Yaskawa INFORM job: OK_R2_O26(120,90)POSPAWANE.JBI

/JOB
//NAME OK_R2_O26(120,90)POSPAWANE
///FOLDERNAME X4
//POS
///NPOS 76,76,76,3,0,0
///TOOL 0
///POSTYPE PULSE
///PULSE
C00000=-124687,-83177,-100814,4913,99770,76656
C00001=-124710,-87372,-98535,4861,96226,76509
C00002=-124720,-88823,-97522,4846,94862,76452
C00003=-124678,-87356,-95828,4839,94572,76455
C00004=-124720,-88823,-97522,4846,94862,76452
C00005=-94650,-94699,-99032,-20051,93372,70764
C00006=-96283,-95826,-99477,-19873,92695,70300
C00007=-94650,-94699,-99032,-20051,93372,70764
C00008=-127024,-94781,-101034,6932,94604,73639
C00009=-125486,-94406,-100478,6779,94328,74137
C00010=-125580,-97568,-101093,6774,93098,74039
C00011=-125486,-94406,-100478,6779,94328,74137
C00012=-127024,-94781,-101034,6932,94604,73639
C00013=-126741,-87687,-96957,6922,95710,73795
C00014=-126718,-86230,-97962,6944,97065,73878
C00015=-126662,-82027,-100223,7023,100586,74095
C00016=-123675,-116589,-109803,7997,69973,-81393
C00017=-122744,-114748,-105092,7760,67947,-81192
C00018=-122375,-113926,-103174,7667,67160,-81109
C00019=-124288,-113805,-103134,8357,67388,-81794
C00020=-124245,-111702,-101340,8343,67360,-81780
C00021=-124288,-113805,-103134,8357,67388,-81794
C00022=-122375,-113926,-103174,7667,67160,-81109
C00023=-138630,-81193,-91554,22902,91021,-82706
C00024=-137093,-81891,-91862,22646,90453,-82269
C00025=-138630,-81193,-91554,22902,91021,-82706
C00026=-138527,-80465,-90405,22879,90685,-82733
C00027=-99714,-84314,-92829,-14326,90379,-83348
C00028=-99332,-87085,-93392,-14378,89399,-83105
C00029=-99714,-84314,-92829,-14326,90379,-83348
C00030=-100119,-76546,-91010,-14307,93097,-83800
C00031=-99872,-75926,-91520,-14362,93752,-83793
C00032=-120615,-96879,-94500,12422,61763,-56469
C00033=-120615,-96444,-91045,12645,59903,-56681
C00034=-120614,-96198,-89632,12739,59177,-56766
C00035=-120612,-97964,-91396,12715,59351,-56744
C00036=-122358,-96168,-89622,13602,59468,-57423
C00037=-120614,-96100,-89110,12773,58912,-56797
C00038=-120614,-95936,-88283,12829,58498,-56846
C00039=-120614,-95844,-87846,12859,58281,-56872
C00040=-120614,-95993,-88552,13310,59748,-59437
C00041=-120614,-96276,-90020,13213,60486,-59348
C00042=-120615,-96798,-93612,12981,62380,-59123
C00043=-120616,-96853,-99747,5843,73141,-72527
C00044=-120615,-96881,-95746,5920,70677,-72647
C00045=-120615,-96762,-94095,5954,69726,-72694
C00046=-120646,-98510,-95846,5959,69908,-72696
C00047=-120787,-94368,-93966,5976,70884,-72697
C00048=-120615,-96784,-94531,4240,70392,-75290
C00049=-120615,-96741,-94529,-89,69852,-81815
C00050=-120615,-96737,-94499,-2085,69975,-84977
C00051=-120615,-96736,-94490,-2287,69985,-85289
C00052=-120615,-96833,-96173,-2273,70970,-85308
C00053=-120616,-96725,-100243,-2243,73529,-85356
C00054=-120616,-95180,-99735,-2469,75570,69309
C00055=-120615,-95387,-95787,-2498,73036,69361
C00056=-120615,-95334,-94154,-2510,72060,69381
C00057=-120451,-92546,-93661,-2552,73193,69414
C00058=-120612,-97039,-95899,-2509,72258,69378
C00059=-120615,-95352,-94373,-2037,72369,71923
C00060=-120615,-95364,-94077,-88,70775,81896
C00061=-120615,-95363,-94184,611,71183,86811
C00062=-120615,-95363,-94196,663,71233,87105
C00063=-120615,-95421,-95866,660,72230,87111
C00064=-120616,-95208,-99899,652,74822,87124
C00065=-120615,-95299,-94637,-6871,62387,55584
C00066=-120614,-95009,-91097,-7001,60372,55709
C00067=-120614,-94810,-89647,-7055,59587,55759
C00068=-118889,-94770,-89630,-7927,59757,56418
C00069=-120611,-96543,-91406,-7043,59778,55748
C00070=-120614,-94727,-89127,-7075,59312,55777
C00071=-120614,-94586,-88313,-7105,58886,55805
C00072=-120614,-94507,-87881,-7122,58663,55819
C00073=-120614,-94585,-88318,-7722,59518,58470
C00074=-120614,-94829,-89821,-7661,60310,58414
C00075=-120615,-95230,-93492,-7517,62345,58276
BC00000=376622,809313,1075175
BC00001=376622,809313,1075175
BC00002=376622,809313,1075175
BC00003=376622,809313,1075175
BC00004=376622,809313,1075175
BC00005=376622,809313,1075175
BC00006=376622,809313,1075175
BC00007=376622,809313,1075175
BC00008=376622,809313,1075175
BC00009=376622,809313,1075175
BC00010=376622,809313,1075175
BC00011=376622,809313,1075175
BC00012=376622,809313,1075175
BC00013=376622,809313,1075175
BC00014=376622,809313,1075175
BC00015=376622,809313,1075175
BC00016=52273,792808,1075175
BC00017=52273,792808,1075175
BC00018=52273,792808,1075175
BC00019=52273,792808,1075175
BC00020=52273,792808,1075175
BC00021=52273,792808,1075175
BC00022=52273,792808,1075175
BC00023=52273,792808,1075175
BC00024=52273,792808,1075175
BC00025=52273,792808,1075175
BC00026=52273,792808,1075175
BC00027=52273,792808,1075175
BC00028=52273,792808,1075175
BC00029=52273,792808,1075175
BC00030=52273,792808,1075175
BC00031=52273,792808,1075175
BC00032=31139,761154,1075175
BC00033=35098,763884,1075175
BC00034=36682,764976,1075175
BC00035=36682,764976,1075175
BC00036=36682,764976,1075175
BC00037=36681,763425,1075175
BC00038=36680,760983,1075175
BC00039=36680,759697,1075175
BC00040=36055,761766,1075175
BC00041=34507,760803,1075175
BC00042=30635,758395,1075175
BC00043=47521,773064,1075175
BC00044=49344,773907,1075175
BC00045=50073,774244,1075175
BC00046=50073,774244,1075175
BC00047=50073,774244,1075175
BC00048=53791,775068,1075175
BC00049=63690,774133,1075175
BC00050=64051,774302,1075175
BC00051=64091,774316,1075175
BC00052=64372,774025,1075175
BC00053=65074,773297,1075175
BC00054=385972,775396,1075175
BC00055=384263,776174,1075175
BC00056=383580,776486,1075175
BC00057=383580,776486,1075175
BC00058=383580,776486,1075175
BC00059=382014,777113,1075175
BC00060=375597,775186,1075175
BC00061=377262,775741,1075175
BC00062=377349,775806,1075175
BC00063=377075,775542,1075175
BC00064=376388,774882,1075175
BC00065=397120,759651,1075175
BC00066=393760,762530,1075175
BC00067=392415,763682,1075175
BC00068=392415,763682,1075175
BC00069=392415,763682,1075175
BC00070=392416,762121,1075175
BC00071=392417,759689,1075175
BC00072=392418,758406,1075175
BC00073=393152,759706,1075175
BC00074=394462,758663,1075175
BC00075=397738,756055,1075175
EC00000=1064209,556475
EC00001=1064209,556475
EC00002=1064209,556475
EC00003=1064209,556475
EC00004=1064209,556475
EC00005=1064209,556475
EC00006=1064209,556475
EC00007=1064209,556475
EC00008=1064209,556475
EC00009=1064209,556475
EC00010=1064209,556475
EC00011=1064209,556475
EC00012=1064209,556475
EC00013=1064209,556475
EC00014=1064209,556475
EC00015=1064209,556475
EC00016=1064209,556475
EC00017=1064209,556475
EC00018=1064209,556475
EC00019=1064209,556475
EC00020=1064209,556475
EC00021=1064209,556475
EC00022=1064209,556475
EC00023=1064209,556475
EC00024=1064209,556475
EC00025=1064209,556475
EC00026=1064209,556475
EC00027=1064209,556475
EC00028=1064209,556475
EC00029=1064209,556475
EC00030=1064209,556475
EC00031=1064209,556475
EC00032=1064209,556475
EC00033=1064209,556475
EC00034=1064209,556475
EC00035=1064209,556475
EC00036=1064209,556475
EC00037=1064209,556475
EC00038=1064209,556475
EC00039=1064209,556475
EC00040=1064209,556475
EC00041=1064209,556475
EC00042=1064209,556475
EC00043=1064209,556475
EC00044=1064209,556475
EC00045=1064209,556475
EC00046=1064209,556475
EC00047=1064209,556475
EC00048=1064209,556475
EC00049=1064209,556475
EC00050=1064209,556475
EC00051=1064209,556475
EC00052=1064209,556475
EC00053=1064209,556475
EC00054=1064209,556475
EC00055=1064209,556475
EC00056=1064209,556475
EC00057=1064209,556475
EC00058=1064209,556475
EC00059=1064209,556475
EC00060=1064209,556475
EC00061=1064209,556475
EC00062=1064209,556475
EC00063=1064209,556475
EC00064=1064209,556475
EC00065=1064209,556475
EC00066=1064209,556475
EC00067=1064209,556475
EC00068=1064209,556475
EC00069=1064209,556475
EC00070=1064209,556475
EC00071=1064209,556475
EC00072=1064209,556475
EC00073=1064209,556475
EC00074=1064209,556475
EC00075=1064209,556475
///POSTYPE BASE
///RECTAN
///RCONF 0,0,0,0,0,0,0,0,0,0,0,0,0,0,0,0,0,0,0,0,0,0,0,0
P00006=0.222,-3.123,-1.508,0.0000,0.0000,0.0000
P00021=-0.225,-6.128,-0.405,0.0000,0.0000,0.0000
P00022=0.222,-3.123,-1.508,0.0000,0.0000,0.0000
//INST
///DATE 2023/12/13 11:22
///ATTR SC,RW
///GROUP1 RB1,BS1
///GROUP2 ST1
NOP
'OK_r2_O26(120,90)
'Path S1043
SFTOF3D
MOVJ C00000 BC00000 VJ=100.00  +MOVJ EC00000 VJ=100.00
MOVL C00001 BC00001 V=400.0  +MOVJ EC00001 VJ=100.00
SMOVL C00002 BC00002 V=60.0  +MOVJ EC00002
SREFP 3 C00003 BC00003  +REFP EC00003
CALL JOB:SEARCH-R1-S13D
SET P022 P006
SFTON3D P022
SMOVL C00004 BC00004 V=60.0  +MOVJ EC00004
SMOVL C00005 BC00005 V=60.0  +MOVJ EC00005
SREFP 3 C00006 BC00006  +REFP EC00006
CALL JOB:SEARCH-R1-S13D
SET P022 P006
SFTON3D P022
SMOVL C00007 BC00007 V=60.0  +MOVJ EC00007
SMOVL C00008 BC00008 V=100.0  +MOVJ EC00008
SMOVL C00009 BC00009 V=60.0  +MOVJ EC00009
SREFP 3 C00010 BC00010  +REFP EC00010
CALL JOB:SEARCH-R1-S13D
SET P022 P006
SFTON3D P022
SMOVL C00011 BC00011 V=60.0  +MOVJ EC00011
SMOVL C00012 BC00012 V=100.0  +MOVJ EC00012
SMOVL C00013 BC00013 V=100.0  +MOVJ EC00013
MOVL C00014 BC00014 V=400.0  +MOVJ EC00014 VJ=100.00
MOVL C00015 BC00015 V=1000.0  +MOVJ EC00015 VJ=100.00
'Path S1432
SFTOF3D
MOVJ C00016 BC00016 VJ=100.00  +MOVJ EC00016 VJ=100.00
MOVL C00017 BC00017 V=400.0  +MOVJ EC00017 VJ=100.00
SMOVL C00018 BC00018 V=100.0  +MOVJ EC00018
SMOVL C00019 BC00019 V=60.0  +MOVJ EC00019
SREFP 3 C00020 BC00020  +REFP EC00020
CALL JOB:SEARCH-R1-S13D
SET P021 P006
SFTON3D P021
SMOVL C00021 BC00021 V=60.0  +MOVJ EC00021
SMOVL C00022 BC00022 V=100.0  +MOVJ EC00022
SMOVL C00023 BC00023 V=60.0  +MOVJ EC00023
SREFP 3 C00024 BC00024  +REFP EC00024
CALL JOB:SEARCH-R1-S13D
SET P021 P006
SFTON3D P021
SMOVL C00025 BC00025 V=60.0  +MOVJ EC00025
SMOVL C00026 BC00026 V=100.0  +MOVJ EC00026
SMOVL C00027 BC00027 V=60.0  +MOVJ EC00027
SREFP 3 C00028 BC00028  +REFP EC00028
CALL JOB:SEARCH-R1-S13D
SET P021 P006
SFTON3D P021
SMOVL C00029 BC00029 V=60.0  +MOVJ EC00029
SMOVL C00030 BC00030 V=100.0  +MOVJ EC00030
MOVL C00031 BC00031 V=400.0  +MOVJ EC00031 VJ=100.00
'Path W1433
SFTOF3D
SFTON3D P021
MOVJ C00032 BC00032 VJ=100.00  +MOVJ EC00032 VJ=100.00
SMOVL C00033 BC00033 V=100.0  +MOVJ EC00033
SMOVL C00034 BC00034 V=100.0 PL=0  +MOVJ EC00034
SREFP 1 C00035 BC00035  +REFP EC00035
SREFP 2 C00036 BC00036  +REFP EC00036
MACRO1 MJ#(0) ARGF0
ARCON
SMOVL C00037 BC00037 V=10.0  +MOVJ EC00037
SMOVL C00038 BC00038 V=10.0  +MOVJ EC00038
SMOVL C00039 BC00039 V=10.0  +MOVJ EC00039
SMOVL C00040 BC00040 V=10.0  +MOVJ EC00040
ARCOF
SMOVL C00041 BC00041 V=400.0  +MOVJ EC00041
SMOVL C00042 BC00042 V=1000.0  +MOVJ EC00042
SFTOF3D
'Path W1434
SFTOF3D
SFTON3D P021
MOVJ C00043 BC00043 VJ=100.00  +MOVJ EC00043 VJ=100.00
SFTOF3D
MOVL C00044 BC00044 V=100.0  +MOVJ EC00044 VJ=100.00
SMOVL C00045 BC00045 V=100.0 PL=0  +MOVJ EC00045
SREFP 1 C00046 BC00046  +REFP EC00046
SREFP 2 C00047 BC00047  +REFP EC00047
MACRO1 MJ#(0) ARGF0
ARCON
SMOVL C00048 BC00048 V=10.0  +MOVJ EC00048
SMOVL C00049 BC00049 V=10.0  +MOVJ EC00049
SMOVL C00050 BC00050 V=10.0  +MOVJ EC00050
SMOVL C00051 BC00051 V=10.0  +MOVJ EC00051
ARCOF
MOVL C00052 BC00052 V=400.0  +MOVJ EC00052 VJ=100.00
MOVL C00053 BC00053 V=1000.0  +MOVJ EC00053 VJ=100.00
'Path W1042
SFTOF3D
SFTON3D P022
MOVJ C00054 BC00054 VJ=100.00  +MOVJ EC00054 VJ=100.00
SMOVL C00055 BC00055 V=400.0  +MOVJ EC00055
SMOVL C00056 BC00056 V=100.0 PL=0  +MOVJ EC00056
SREFP 1 C00057 BC00057  +REFP EC00057
SREFP 2 C00058 BC00058  +REFP EC00058
MACRO1 MJ#(0) ARGF0
ARCON
SMOVL C00059 BC00059 V=10.0  +MOVJ EC00059
SMOVL C00060 BC00060 V=10.0  +MOVJ EC00060
SMOVL C00061 BC00061 V=10.0  +MOVJ EC00061
SMOVL C00062 BC00062 V=10.0  +MOVJ EC00062
ARCOF
SMOVL C00063 BC00063 V=400.0  +MOVJ EC00063
SMOVL C00064 BC00064 V=1000.0  +MOVJ EC00064
SFTOF3D
'Path W1041
SFTOF3D
SFTON3D P022
MOVJ C00065 BC00065 VJ=100.00  +MOVJ EC00065 VJ=100.00
SMOVL C00066 BC00066 V=400.0  +MOVJ EC00066
SMOVL C00067 BC00067 V=100.0 PL=0  +MOVJ EC00067
SREFP 1 C00068 BC00068  +REFP EC00068
SREFP 2 C00069 BC00069  +REFP EC00069
MACRO1 MJ#(0) ARGF0
ARCON
SMOVL C00070 BC00070 V=10.0  +MOVJ EC00070
SMOVL C00071 BC00071 V=10.0  +MOVJ EC00071
SMOVL C00072 BC00072 V=10.0  +MOVJ EC00072
SMOVL C00073 BC00073 V=10.0  +MOVJ EC00073
ARCOF
SMOVL C00074 BC00074 V=400.0  +MOVJ EC00074
SMOVL C00075 BC00075 V=1000.0  +MOVJ EC00075
SFTOF3D
END
